// Mitsubishi GX Works2 project: 10   PLC: FX2N/FX2NC

PROGRAM MAIN
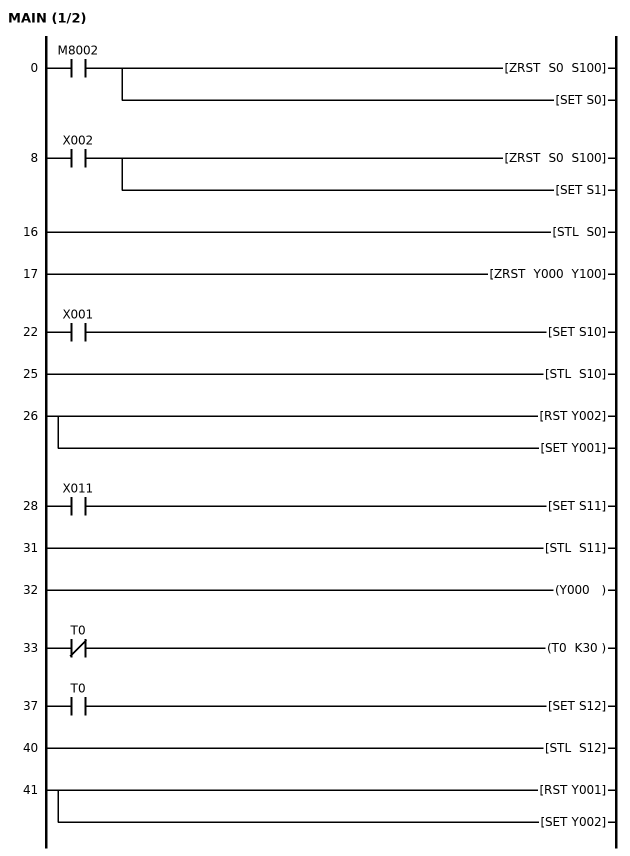
0     LD      M8002
      ZRST    S0 S100
      SET     S0
8     LD      X002
      ZRST    S0 S100
      SET     S1
16    STL     S0
17    ZRST    Y000 Y100
22    LD      X001
      SET     S10
25    STL     S10
26    RST     Y002
      SET     Y001
28    LD      X011
      SET     S11
31    STL     S11
32    OUT     Y000
33    LDI     T0
      OUT     T0 K30
37    LD      T0
      SET     S12
40    STL     S12
41    RST     Y001
      SET     Y002
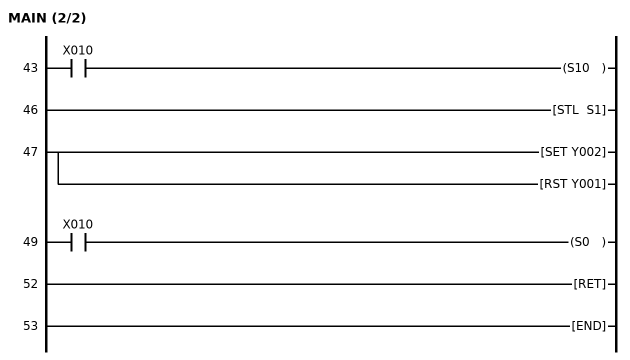
43    LD      X010
      OUT     S10
46    STL     S1
47    SET     Y002
      RST     Y001
49    LD      X010
      OUT     S0
52    RET
53    END
END_PROGRAM

// device comments not shown above
BL0  ; main
BL1  ; a
BL2  ; b
